KUKA KRL program: AM001.src, AM001.dat

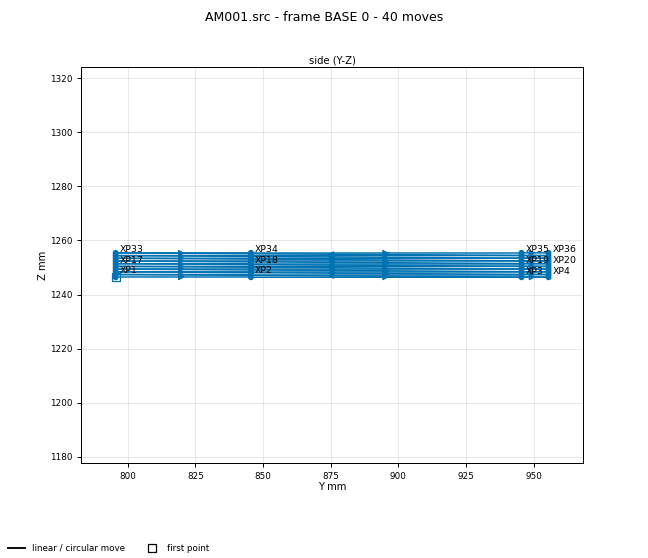
[picture p0: tool path of AM001.src in frame BASE 0, 40 of 42 moves have a stored position in this frame; points joined in program order, loops and branches not executed]
--- AM001.src ---
&ACCESS RVP
&REL 154
&PARAM TEMPLATE = C:\KRC\Roboter\Template\vorgabe
&PARAM EDITMASK = *
DEF AM001( )
;FOLD INI
  ;FOLD BASISTECH INI
    GLOBAL INTERRUPT DECL 3 WHEN $STOPMESS==TRUE DO IR_STOPM ( )
    INTERRUPT ON 3
    BAS (#INITMOV,0 )
  ;ENDFOLD (BASISTECH INI)
  ;FOLD USER INI
    ;Make your modifications here

  ;ENDFOLD (USER INI)
;ENDFOLD (INI)

;FOLD PTP HOME Vel=10 % DEFAULT;%{PE}%R 5.6.13,%MKUKATPBASIS,%CMOVE,%VPTP,%P 1:PTP, 2:HOME, 3:, 5:10, 7:DEFAULT
$BWDSTART=FALSE
PDAT_ACT=PDEFAULT
FDAT_ACT=FHOME
BAS(#PTP_PARAMS,10)
$H_POS=XHOME
PTP XHOME
;ENDFOLD

;FOLD OUT 33 'Gas 1' State=TRUE CONT;%{PE}%R 5.6.13,%MKUKATPBASIS,%COUT,%VOUTX,%P 2:33, 3:Gas 1, 5:TRUE, 6:CONTINUE
CONTINUE
$OUT[33]=TRUE
;ENDFOLD
;FOLD OUT 36 'Gas 2' State=TRUE CONT;%{PE}%R 5.6.13,%MKUKATPBASIS,%COUT,%VOUTX,%P 2:36, 3:Gas 2, 5:TRUE, 6:CONTINUE
CONTINUE
$OUT[36]=TRUE
;ENDFOLD
;FOLD WAIT Time=3 sec;%{PE}%R 5.6.13,%MKUKATPBASIS,%CWAIT,%VWAIT,%P 2:3
WAIT SEC 3
;ENDFOLD
;FOLD ANOUT POWDER=0.2 ;%{PE}%R 5.6.13,%MKUKATPBASIS,%CANA,%VANOUT_STAT,%P 2:CHANNEL_1, 4:0.2
$ANOUT[1]=0.2
;ENDFOLD
;FOLD LIN P1 Vel=0.035 m/s CPDAT1 Tool[1] Base[0];%{PE}%R 5.6.13,%MKUKATPBASIS,%CMOVE,%VLIN,%P 1:LIN, 2:P1, 3:, 5:0.035, 7:CPDAT1
$BWDSTART=FALSE
LDAT_ACT=LCPDAT1
FDAT_ACT=FP1
BAS(#CP_PARAMS,0.035)
LIN XP1
;ENDFOLD
;FOLD LIN P2 CONT Vel=0.035 m/s CPDAT2 Tool[1] Base[0];%{PE}%R 5.6.13,%MKUKATPBASIS,%CMOVE,%VLIN,%P 1:LIN, 2:P2, 3:C_DIS, 5:0.035, 7:CPDAT2
$BWDSTART=FALSE
LDAT_ACT=LCPDAT2
FDAT_ACT=FP2
BAS(#CP_PARAMS,0.035)
LIN XP2 C_DIS
;ENDFOLD
;FOLD SYN OUT 34 'Laser Shutter' State=TRUE at START Delay=0 ms;%{PE}%R 5.6.13,%MKUKATPBASIS,%COUT,%VSYNOUT,%P 2:34, 3:Laser Shutter, 5:TRUE, 7:0, 9:0, 12:0
TRIGGER WHEN DISTANCE=0 DELAY=0 DO $OUT[34]=TRUE
;ENDFOLD
;FOLD LIN P3 CONT Vel=0.035 m/s CPDAT3 Tool[1] Base[0];%{PE}%R 5.6.13,%MKUKATPBASIS,%CMOVE,%VLIN,%P 1:LIN, 2:P3, 3:C_DIS, 5:0.035, 7:CPDAT3
$BWDSTART=FALSE
LDAT_ACT=LCPDAT3
FDAT_ACT=FP3
BAS(#CP_PARAMS,0.035)
LIN XP3 C_DIS
;ENDFOLD
;FOLD SYN OUT 34 'Laser Shutter' State=FALSE at START Delay=0 ms;%{PE}%R 5.6.13,%MKUKATPBASIS,%COUT,%VSYNOUT,%P 2:34, 3:Laser Shutter, 5:FALSE, 7:0, 9:0, 12:0
TRIGGER WHEN DISTANCE=0 DELAY=0 DO $OUT[34]=FALSE
;ENDFOLD
;FOLD ANOUT POWDER=0 ;%{PE}%R 5.6.13,%MKUKATPBASIS,%CANA,%VANOUT_STAT,%P 2:CHANNEL_1, 4:0
$ANOUT[1]=0
;ENDFOLD
;FOLD LIN P4 Vel=0.035 m/s CPDAT4 Tool[1] Base[0];%{PE}%R 5.6.13,%MKUKATPBASIS,%CMOVE,%VLIN,%P 1:LIN, 2:P4, 3:, 5:0.035, 7:CPDAT4
$BWDSTART=FALSE
LDAT_ACT=LCPDAT4
FDAT_ACT=FP4
BAS(#CP_PARAMS,0.035)
LIN XP4
;ENDFOLD
;FOLD WAIT Time=0.1 sec;%{PE}%R 5.6.13,%MKUKATPBASIS,%CWAIT,%VWAIT,%P 2:0.1
WAIT SEC 0.1
;ENDFOLD
;FOLD ANOUT POWDER=0.2 ;%{PE}%R 5.6.13,%MKUKATPBASIS,%CANA,%VANOUT_STAT,%P 2:CHANNEL_1, 4:0.2
$ANOUT[1]=0.2
;ENDFOLD
;FOLD LIN P5 Vel=0.035 m/s CPDAT5 Tool[1] Base[0];%{PE}%R 5.6.13,%MKUKATPBASIS,%CMOVE,%VLIN,%P 1:LIN, 2:P5, 3:, 5:0.035, 7:CPDAT5
$BWDSTART=FALSE
LDAT_ACT=LCPDAT5
FDAT_ACT=FP5
BAS(#CP_PARAMS,0.035)
LIN XP5
;ENDFOLD
;FOLD LIN P6 CONT Vel=0.035 m/s CPDAT6 Tool[1] Base[0];%{PE}%R 5.6.13,%MKUKATPBASIS,%CMOVE,%VLIN,%P 1:LIN, 2:P6, 3:C_DIS, 5:0.035, 7:CPDAT6
$BWDSTART=FALSE
LDAT_ACT=LCPDAT6
FDAT_ACT=FP6
BAS(#CP_PARAMS,0.035)
LIN XP6 C_DIS
;ENDFOLD
;FOLD SYN OUT 34 'Laser Shutter' State=TRUE at START Delay=0 ms;%{PE}%R 5.6.13,%MKUKATPBASIS,%COUT,%VSYNOUT,%P 2:34, 3:Laser Shutter, 5:TRUE, 7:0, 9:0, 12:0
TRIGGER WHEN DISTANCE=0 DELAY=0 DO $OUT[34]=TRUE
;ENDFOLD
;FOLD LIN P7 CONT Vel=0.035 m/s CPDAT7 Tool[1] Base[0];%{PE}%R 5.6.13,%MKUKATPBASIS,%CMOVE,%VLIN,%P 1:LIN, 2:P7, 3:C_DIS, 5:0.035, 7:CPDAT7
$BWDSTART=FALSE
LDAT_ACT=LCPDAT7
FDAT_ACT=FP7
BAS(#CP_PARAMS,0.035)
LIN XP7 C_DIS
;ENDFOLD
;FOLD SYN OUT 34 'Laser Shutter' State=FALSE at START Delay=0 ms;%{PE}%R 5.6.13,%MKUKATPBASIS,%COUT,%VSYNOUT,%P 2:34, 3:Laser Shutter, 5:FALSE, 7:0, 9:0, 12:0
TRIGGER WHEN DISTANCE=0 DELAY=0 DO $OUT[34]=FALSE
;ENDFOLD
;FOLD ANOUT POWDER=0 ;%{PE}%R 5.6.13,%MKUKATPBASIS,%CANA,%VANOUT_STAT,%P 2:CHANNEL_1, 4:0
$ANOUT[1]=0
;ENDFOLD
;FOLD LIN P8 Vel=0.035 m/s CPDAT8 Tool[1] Base[0];%{PE}%R 5.6.13,%MKUKATPBASIS,%CMOVE,%VLIN,%P 1:LIN, 2:P8, 3:, 5:0.035, 7:CPDAT8
$BWDSTART=FALSE
LDAT_ACT=LCPDAT8
FDAT_ACT=FP8
BAS(#CP_PARAMS,0.035)
LIN XP8
;ENDFOLD
;FOLD WAIT Time=0.1 sec;%{PE}%R 5.6.13,%MKUKATPBASIS,%CWAIT,%VWAIT,%P 2:0.1
WAIT SEC 0.1
;ENDFOLD
;FOLD ANOUT POWDER=0.2 ;%{PE}%R 5.6.13,%MKUKATPBASIS,%CANA,%VANOUT_STAT,%P 2:CHANNEL_1, 4:0.2
$ANOUT[1]=0.2
;ENDFOLD
;FOLD LIN P9 Vel=0.035 m/s CPDAT9 Tool[1] Base[0];%{PE}%R 5.6.13,%MKUKATPBASIS,%CMOVE,%VLIN,%P 1:LIN, 2:P9, 3:, 5:0.035, 7:CPDAT9
$BWDSTART=FALSE
LDAT_ACT=LCPDAT9
FDAT_ACT=FP9
BAS(#CP_PARAMS,0.035)
LIN XP9
;ENDFOLD
;FOLD LIN P10 CONT Vel=0.035 m/s CPDAT10 Tool[1] Base[0];%{PE}%R 5.6.13,%MKUKATPBASIS,%CMOVE,%VLIN,%P 1:LIN, 2:P10, 3:C_DIS, 5:0.035, 7:CPDAT10
$BWDSTART=FALSE
LDAT_ACT=LCPDAT10
FDAT_ACT=FP10
BAS(#CP_PARAMS,0.035)
LIN XP10 C_DIS
;ENDFOLD
;FOLD SYN OUT 34 'Laser Shutter' State=TRUE at START Delay=0 ms;%{PE}%R 5.6.13,%MKUKATPBASIS,%COUT,%VSYNOUT,%P 2:34, 3:Laser Shutter, 5:TRUE, 7:0, 9:0, 12:0
TRIGGER WHEN DISTANCE=0 DELAY=0 DO $OUT[34]=TRUE
;ENDFOLD
;FOLD LIN P11 CONT Vel=0.035 m/s CPDAT11 Tool[1] Base[0];%{PE}%R 5.6.13,%MKUKATPBASIS,%CMOVE,%VLIN,%P 1:LIN, 2:P11, 3:C_DIS, 5:0.035, 7:CPDAT11
$BWDSTART=FALSE
LDAT_ACT=LCPDAT11
FDAT_ACT=FP11
BAS(#CP_PARAMS,0.035)
LIN XP11 C_DIS
;ENDFOLD
;FOLD SYN OUT 34 'Laser Shutter' State=FALSE at START Delay=0 ms;%{PE}%R 5.6.13,%MKUKATPBASIS,%COUT,%VSYNOUT,%P 2:34, 3:Laser Shutter, 5:FALSE, 7:0, 9:0, 12:0
TRIGGER WHEN DISTANCE=0 DELAY=0 DO $OUT[34]=FALSE
;ENDFOLD
;FOLD ANOUT POWDER=0 ;%{PE}%R 5.6.13,%MKUKATPBASIS,%CANA,%VANOUT_STAT,%P 2:CHANNEL_1, 4:0
$ANOUT[1]=0
;ENDFOLD
;FOLD LIN P12 Vel=0.035 m/s CPDAT12 Tool[1] Base[0];%{PE}%R 5.6.13,%MKUKATPBASIS,%CMOVE,%VLIN,%P 1:LIN, 2:P12, 3:, 5:0.035, 7:CPDAT12
$BWDSTART=FALSE
LDAT_ACT=LCPDAT12
FDAT_ACT=FP12
BAS(#CP_PARAMS,0.035)
LIN XP12
;ENDFOLD
;FOLD WAIT Time=0.1 sec;%{PE}%R 5.6.13,%MKUKATPBASIS,%CWAIT,%VWAIT,%P 2:0.1
WAIT SEC 0.1
;ENDFOLD
;FOLD ANOUT POWDER=0.2 ;%{PE}%R 5.6.13,%MKUKATPBASIS,%CANA,%VANOUT_STAT,%P 2:CHANNEL_1, 4:0.2
$ANOUT[1]=0.2
;ENDFOLD
;FOLD LIN P13 Vel=0.035 m/s CPDAT13 Tool[1] Base[0];%{PE}%R 5.6.13,%MKUKATPBASIS,%CMOVE,%VLIN,%P 1:LIN, 2:P13, 3:, 5:0.035, 7:CPDAT13
$BWDSTART=FALSE
LDAT_ACT=LCPDAT13
FDAT_ACT=FP13
BAS(#CP_PARAMS,0.035)
LIN XP13
;ENDFOLD
;FOLD LIN P14 CONT Vel=0.035 m/s CPDAT14 Tool[1] Base[0];%{PE}%R 5.6.13,%MKUKATPBASIS,%CMOVE,%VLIN,%P 1:LIN, 2:P14, 3:C_DIS, 5:0.035, 7:CPDAT14
$BWDSTART=FALSE
LDAT_ACT=LCPDAT14
FDAT_ACT=FP14
BAS(#CP_PARAMS,0.035)
LIN XP14 C_DIS
;ENDFOLD
;FOLD SYN OUT 34 'Laser Shutter' State=TRUE at START Delay=0 ms;%{PE}%R 5.6.13,%MKUKATPBASIS,%COUT,%VSYNOUT,%P 2:34, 3:Laser Shutter, 5:TRUE, 7:0, 9:0, 12:0
TRIGGER WHEN DISTANCE=0 DELAY=0 DO $OUT[34]=TRUE
;ENDFOLD
;FOLD LIN P15 CONT Vel=0.035 m/s CPDAT15 Tool[1] Base[0];%{PE}%R 5.6.13,%MKUKATPBASIS,%CMOVE,%VLIN,%P 1:LIN, 2:P15, 3:C_DIS, 5:0.035, 7:CPDAT15
$BWDSTART=FALSE
LDAT_ACT=LCPDAT15
FDAT_ACT=FP15
BAS(#CP_PARAMS,0.035)
LIN XP15 C_DIS
;ENDFOLD
;FOLD SYN OUT 34 'Laser Shutter' State=FALSE at START Delay=0 ms;%{PE}%R 5.6.13,%MKUKATPBASIS,%COUT,%VSYNOUT,%P 2:34, 3:Laser Shutter, 5:FALSE, 7:0, 9:0, 12:0
TRIGGER WHEN DISTANCE=0 DELAY=0 DO $OUT[34]=FALSE
;ENDFOLD
;FOLD ANOUT POWDER=0 ;%{PE}%R 5.6.13,%MKUKATPBASIS,%CANA,%VANOUT_STAT,%P 2:CHANNEL_1, 4:0
$ANOUT[1]=0
;ENDFOLD
;FOLD LIN P16 Vel=0.035 m/s CPDAT16 Tool[1] Base[0];%{PE}%R 5.6.13,%MKUKATPBASIS,%CMOVE,%VLIN,%P 1:LIN, 2:P16, 3:, 5:0.035, 7:CPDAT16
$BWDSTART=FALSE
LDAT_ACT=LCPDAT16
FDAT_ACT=FP16
BAS(#CP_PARAMS,0.035)
LIN XP16
;ENDFOLD
;FOLD WAIT Time=0.1 sec;%{PE}%R 5.6.13,%MKUKATPBASIS,%CWAIT,%VWAIT,%P 2:0.1
WAIT SEC 0.1
;ENDFOLD
;FOLD ANOUT POWDER=0.2 ;%{PE}%R 5.6.13,%MKUKATPBASIS,%CANA,%VANOUT_STAT,%P 2:CHANNEL_1, 4:0.2
$ANOUT[1]=0.2
;ENDFOLD
;FOLD LIN P17 Vel=0.035 m/s CPDAT17 Tool[1] Base[0];%{PE}%R 5.6.13,%MKUKATPBASIS,%CMOVE,%VLIN,%P 1:LIN, 2:P17, 3:, 5:0.035, 7:CPDAT17
$BWDSTART=FALSE
LDAT_ACT=LCPDAT17
FDAT_ACT=FP17
BAS(#CP_PARAMS,0.035)
LIN XP17
;ENDFOLD
;FOLD LIN P18 CONT Vel=0.035 m/s CPDAT18 Tool[1] Base[0];%{PE}%R 5.6.13,%MKUKATPBASIS,%CMOVE,%VLIN,%P 1:LIN, 2:P18, 3:C_DIS, 5:0.035, 7:CPDAT18
$BWDSTART=FALSE
LDAT_ACT=LCPDAT18
FDAT_ACT=FP18
BAS(#CP_PARAMS,0.035)
LIN XP18 C_DIS
;ENDFOLD
;FOLD SYN OUT 34 'Laser Shutter' State=TRUE at START Delay=0 ms;%{PE}%R 5.6.13,%MKUKATPBASIS,%COUT,%VSYNOUT,%P 2:34, 3:Laser Shutter, 5:TRUE, 7:0, 9:0, 12:0
TRIGGER WHEN DISTANCE=0 DELAY=0 DO $OUT[34]=TRUE
;ENDFOLD
;FOLD LIN P19 CONT Vel=0.035 m/s CPDAT19 Tool[1] Base[0];%{PE}%R 5.6.13,%MKUKATPBASIS,%CMOVE,%VLIN,%P 1:LIN, 2:P19, 3:C_DIS, 5:0.035, 7:CPDAT19
$BWDSTART=FALSE
LDAT_ACT=LCPDAT19
FDAT_ACT=FP19
BAS(#CP_PARAMS,0.035)
LIN XP19 C_DIS
;ENDFOLD
;FOLD SYN OUT 34 'Laser Shutter' State=FALSE at START Delay=0 ms;%{PE}%R 5.6.13,%MKUKATPBASIS,%COUT,%VSYNOUT,%P 2:34, 3:Laser Shutter, 5:FALSE, 7:0, 9:0, 12:0
TRIGGER WHEN DISTANCE=0 DELAY=0 DO $OUT[34]=FALSE
;ENDFOLD
;FOLD ANOUT POWDER=0 ;%{PE}%R 5.6.13,%MKUKATPBASIS,%CANA,%VANOUT_STAT,%P 2:CHANNEL_1, 4:0
$ANOUT[1]=0
;ENDFOLD
;FOLD LIN P20 Vel=0.035 m/s CPDAT20 Tool[1] Base[0];%{PE}%R 5.6.13,%MKUKATPBASIS,%CMOVE,%VLIN,%P 1:LIN, 2:P20, 3:, 5:0.035, 7:CPDAT20
$BWDSTART=FALSE
LDAT_ACT=LCPDAT20
FDAT_ACT=FP20
BAS(#CP_PARAMS,0.035)
LIN XP20
;ENDFOLD
;FOLD WAIT Time=0.1 sec;%{PE}%R 5.6.13,%MKUKATPBASIS,%CWAIT,%VWAIT,%P 2:0.1
WAIT SEC 0.1
;ENDFOLD
;FOLD ANOUT POWDER=0.2 ;%{PE}%R 5.6.13,%MKUKATPBASIS,%CANA,%VANOUT_STAT,%P 2:CHANNEL_1, 4:0.2
$ANOUT[1]=0.2
;ENDFOLD
;FOLD LIN P21 Vel=0.035 m/s CPDAT21 Tool[1] Base[0];%{PE}%R 5.6.13,%MKUKATPBASIS,%CMOVE,%VLIN,%P 1:LIN, 2:P21, 3:, 5:0.035, 7:CPDAT21
$BWDSTART=FALSE
LDAT_ACT=LCPDAT21
FDAT_ACT=FP21
BAS(#CP_PARAMS,0.035)
LIN XP21
;ENDFOLD
;FOLD LIN P22 CONT Vel=0.035 m/s CPDAT22 Tool[1] Base[0];%{PE}%R 5.6.13,%MKUKATPBASIS,%CMOVE,%VLIN,%P 1:LIN, 2:P22, 3:C_DIS, 5:0.035, 7:CPDAT22
$BWDSTART=FALSE
LDAT_ACT=LCPDAT22
FDAT_ACT=FP22
BAS(#CP_PARAMS,0.035)
LIN XP22 C_DIS
;ENDFOLD
;FOLD SYN OUT 34 'Laser Shutter' State=TRUE at START Delay=0 ms;%{PE}%R 5.6.13,%MKUKATPBASIS,%COUT,%VSYNOUT,%P 2:34, 3:Laser Shutter, 5:TRUE, 7:0, 9:0, 12:0
TRIGGER WHEN DISTANCE=0 DELAY=0 DO $OUT[34]=TRUE
;ENDFOLD
;FOLD LIN P23 CONT Vel=0.035 m/s CPDAT23 Tool[1] Base[0];%{PE}%R 5.6.13,%MKUKATPBASIS,%CMOVE,%VLIN,%P 1:LIN, 2:P23, 3:C_DIS, 5:0.035, 7:CPDAT23
$BWDSTART=FALSE
LDAT_ACT=LCPDAT23
FDAT_ACT=FP23
BAS(#CP_PARAMS,0.035)
LIN XP23 C_DIS
;ENDFOLD
;FOLD SYN OUT 34 'Laser Shutter' State=FALSE at START Delay=0 ms;%{PE}%R 5.6.13,%MKUKATPBASIS,%COUT,%VSYNOUT,%P 2:34, 3:Laser Shutter, 5:FALSE, 7:0, 9:0, 12:0
TRIGGER WHEN DISTANCE=0 DELAY=0 DO $OUT[34]=FALSE
;ENDFOLD
;FOLD ANOUT POWDER=0 ;%{PE}%R 5.6.13,%MKUKATPBASIS,%CANA,%VANOUT_STAT,%P 2:CHANNEL_1, 4:0
$ANOUT[1]=0
;ENDFOLD
;FOLD LIN P24 Vel=0.035 m/s CPDAT24 Tool[1] Base[0];%{PE}%R 5.6.13,%MKUKATPBASIS,%CMOVE,%VLIN,%P 1:LIN, 2:P24, 3:, 5:0.035, 7:CPDAT24
$BWDSTART=FALSE
LDAT_ACT=LCPDAT24
FDAT_ACT=FP24
BAS(#CP_PARAMS,0.035)
LIN XP24
;ENDFOLD
;FOLD WAIT Time=0.1 sec;%{PE}%R 5.6.13,%MKUKATPBASIS,%CWAIT,%VWAIT,%P 2:0.1
WAIT SEC 0.1
;ENDFOLD
;FOLD ANOUT POWDER=0.2 ;%{PE}%R 5.6.13,%MKUKATPBASIS,%CANA,%VANOUT_STAT,%P 2:CHANNEL_1, 4:0.2
$ANOUT[1]=0.2
;ENDFOLD
;FOLD LIN P25 Vel=0.035 m/s CPDAT25 Tool[1] Base[0];%{PE}%R 5.6.13,%MKUKATPBASIS,%CMOVE,%VLIN,%P 1:LIN, 2:P25, 3:, 5:0.035, 7:CPDAT25
$BWDSTART=FALSE
LDAT_ACT=LCPDAT25
FDAT_ACT=FP25
BAS(#CP_PARAMS,0.035)
LIN XP25
;ENDFOLD
;FOLD LIN P26 CONT Vel=0.035 m/s CPDAT26 Tool[1] Base[0];%{PE}%R 5.6.13,%MKUKATPBASIS,%CMOVE,%VLIN,%P 1:LIN, 2:P26, 3:C_DIS, 5:0.035, 7:CPDAT26
$BWDSTART=FALSE
LDAT_ACT=LCPDAT26
FDAT_ACT=FP26
BAS(#CP_PARAMS,0.035)
LIN XP26 C_DIS
;ENDFOLD
;FOLD SYN OUT 34 'Laser Shutter' State=TRUE at START Delay=0 ms;%{PE}%R 5.6.13,%MKUKATPBASIS,%COUT,%VSYNOUT,%P 2:34, 3:Laser Shutter, 5:TRUE, 7:0, 9:0, 12:0
TRIGGER WHEN DISTANCE=0 DELAY=0 DO $OUT[34]=TRUE
;ENDFOLD
;FOLD LIN P27 CONT Vel=0.035 m/s CPDAT27 Tool[1] Base[0];%{PE}%R 5.6.13,%MKUKATPBASIS,%CMOVE,%VLIN,%P 1:LIN, 2:P27, 3:C_DIS, 5:0.035, 7:CPDAT27
$BWDSTART=FALSE
LDAT_ACT=LCPDAT27
FDAT_ACT=FP27
BAS(#CP_PARAMS,0.035)
LIN XP27 C_DIS
;ENDFOLD
;FOLD SYN OUT 34 'Laser Shutter' State=FALSE at START Delay=0 ms;%{PE}%R 5.6.13,%MKUKATPBASIS,%COUT,%VSYNOUT,%P 2:34, 3:Laser Shutter, 5:FALSE, 7:0, 9:0, 12:0
TRIGGER WHEN DISTANCE=0 DELAY=0 DO $OUT[34]=FALSE
;ENDFOLD
;FOLD ANOUT POWDER=0 ;%{PE}%R 5.6.13,%MKUKATPBASIS,%CANA,%VANOUT_STAT,%P 2:CHANNEL_1, 4:0
$ANOUT[1]=0
;ENDFOLD
;FOLD LIN P28 Vel=0.035 m/s CPDAT28 Tool[1] Base[0];%{PE}%R 5.6.13,%MKUKATPBASIS,%CMOVE,%VLIN,%P 1:LIN, 2:P28, 3:, 5:0.035, 7:CPDAT28
$BWDSTART=FALSE
LDAT_ACT=LCPDAT28
FDAT_ACT=FP28
BAS(#CP_PARAMS,0.035)
LIN XP28
;ENDFOLD
;FOLD WAIT Time=0.1 sec;%{PE}%R 5.6.13,%MKUKATPBASIS,%CWAIT,%VWAIT,%P 2:0.1
WAIT SEC 0.1
;ENDFOLD
;FOLD ANOUT POWDER=0.2 ;%{PE}%R 5.6.13,%MKUKATPBASIS,%CANA,%VANOUT_STAT,%P 2:CHANNEL_1, 4:0.2
$ANOUT[1]=0.2
;ENDFOLD
;FOLD LIN P29 Vel=0.035 m/s CPDAT29 Tool[1] Base[0];%{PE}%R 5.6.13,%MKUKATPBASIS,%CMOVE,%VLIN,%P 1:LIN, 2:P29, 3:, 5:0.035, 7:CPDAT29
$BWDSTART=FALSE
LDAT_ACT=LCPDAT29
FDAT_ACT=FP29
BAS(#CP_PARAMS,0.035)
LIN XP29
;ENDFOLD
;FOLD LIN P30 CONT Vel=0.035 m/s CPDAT30 Tool[1] Base[0];%{PE}%R 5.6.13,%MKUKATPBASIS,%CMOVE,%VLIN,%P 1:LIN, 2:P30, 3:C_DIS, 5:0.035, 7:CPDAT30
$BWDSTART=FALSE
LDAT_ACT=LCPDAT30
FDAT_ACT=FP30
BAS(#CP_PARAMS,0.035)
LIN XP30 C_DIS
;ENDFOLD
;FOLD SYN OUT 34 'Laser Shutter' State=TRUE at START Delay=0 ms;%{PE}%R 5.6.13,%MKUKATPBASIS,%COUT,%VSYNOUT,%P 2:34, 3:Laser Shutter, 5:TRUE, 7:0, 9:0, 12:0
TRIGGER WHEN DISTANCE=0 DELAY=0 DO $OUT[34]=TRUE
;ENDFOLD
;FOLD LIN P31 CONT Vel=0.035 m/s CPDAT31 Tool[1] Base[0];%{PE}%R 5.6.13,%MKUKATPBASIS,%CMOVE,%VLIN,%P 1:LIN, 2:P31, 3:C_DIS, 5:0.035, 7:CPDAT31
$BWDSTART=FALSE
LDAT_ACT=LCPDAT31
FDAT_ACT=FP31
BAS(#CP_PARAMS,0.035)
LIN XP31 C_DIS
;ENDFOLD
;FOLD SYN OUT 34 'Laser Shutter' State=FALSE at START Delay=0 ms;%{PE}%R 5.6.13,%MKUKATPBASIS,%COUT,%VSYNOUT,%P 2:34, 3:Laser Shutter, 5:FALSE, 7:0, 9:0, 12:0
TRIGGER WHEN DISTANCE=0 DELAY=0 DO $OUT[34]=FALSE
;ENDFOLD
;FOLD ANOUT POWDER=0 ;%{PE}%R 5.6.13,%MKUKATPBASIS,%CANA,%VANOUT_STAT,%P 2:CHANNEL_1, 4:0
$ANOUT[1]=0
;ENDFOLD
;FOLD LIN P32 Vel=0.035 m/s CPDAT32 Tool[1] Base[0];%{PE}%R 5.6.13,%MKUKATPBASIS,%CMOVE,%VLIN,%P 1:LIN, 2:P32, 3:, 5:0.035, 7:CPDAT32
$BWDSTART=FALSE
LDAT_ACT=LCPDAT32
FDAT_ACT=FP32
BAS(#CP_PARAMS,0.035)
LIN XP32
;ENDFOLD
;FOLD WAIT Time=0.1 sec;%{PE}%R 5.6.13,%MKUKATPBASIS,%CWAIT,%VWAIT,%P 2:0.1
WAIT SEC 0.1
;ENDFOLD
;FOLD ANOUT POWDER=0.2 ;%{PE}%R 5.6.13,%MKUKATPBASIS,%CANA,%VANOUT_STAT,%P 2:CHANNEL_1, 4:0.2
$ANOUT[1]=0.2
;ENDFOLD
;FOLD LIN P33 Vel=0.035 m/s CPDAT33 Tool[1] Base[0];%{PE}%R 5.6.13,%MKUKATPBASIS,%CMOVE,%VLIN,%P 1:LIN, 2:P33, 3:, 5:0.035, 7:CPDAT33
$BWDSTART=FALSE
LDAT_ACT=LCPDAT33
FDAT_ACT=FP33
BAS(#CP_PARAMS,0.035)
LIN XP33
;ENDFOLD
;FOLD LIN P34 CONT Vel=0.035 m/s CPDAT34 Tool[1] Base[0];%{PE}%R 5.6.13,%MKUKATPBASIS,%CMOVE,%VLIN,%P 1:LIN, 2:P34, 3:C_DIS, 5:0.035, 7:CPDAT34
$BWDSTART=FALSE
LDAT_ACT=LCPDAT34
FDAT_ACT=FP34
BAS(#CP_PARAMS,0.035)
LIN XP34 C_DIS
;ENDFOLD
;FOLD SYN OUT 34 'Laser Shutter' State=TRUE at START Delay=0 ms;%{PE}%R 5.6.13,%MKUKATPBASIS,%COUT,%VSYNOUT,%P 2:34, 3:Laser Shutter, 5:TRUE, 7:0, 9:0, 12:0
TRIGGER WHEN DISTANCE=0 DELAY=0 DO $OUT[34]=TRUE
;ENDFOLD
;FOLD LIN P35 CONT Vel=0.035 m/s CPDAT35 Tool[1] Base[0];%{PE}%R 5.6.13,%MKUKATPBASIS,%CMOVE,%VLIN,%P 1:LIN, 2:P35, 3:C_DIS, 5:0.035, 7:CPDAT35
$BWDSTART=FALSE
LDAT_ACT=LCPDAT35
FDAT_ACT=FP35
BAS(#CP_PARAMS,0.035)
LIN XP35 C_DIS
;ENDFOLD
;FOLD SYN OUT 34 'Laser Shutter' State=FALSE at START Delay=0 ms;%{PE}%R 5.6.13,%MKUKATPBASIS,%COUT,%VSYNOUT,%P 2:34, 3:Laser Shutter, 5:FALSE, 7:0, 9:0, 12:0
TRIGGER WHEN DISTANCE=0 DELAY=0 DO $OUT[34]=FALSE
;ENDFOLD
;FOLD ANOUT POWDER=0 ;%{PE}%R 5.6.13,%MKUKATPBASIS,%CANA,%VANOUT_STAT,%P 2:CHANNEL_1, 4:0
$ANOUT[1]=0
;ENDFOLD
;FOLD LIN P36 Vel=0.035 m/s CPDAT36 Tool[1] Base[0];%{PE}%R 5.6.13,%MKUKATPBASIS,%CMOVE,%VLIN,%P 1:LIN, 2:P36, 3:, 5:0.035, 7:CPDAT36
$BWDSTART=FALSE
LDAT_ACT=LCPDAT36
FDAT_ACT=FP36
BAS(#CP_PARAMS,0.035)
LIN XP36
;ENDFOLD
;FOLD WAIT Time=0.1 sec;%{PE}%R 5.6.13,%MKUKATPBASIS,%CWAIT,%VWAIT,%P 2:0.1
WAIT SEC 0.1
;ENDFOLD
;FOLD ANOUT POWDER=0.2 ;%{PE}%R 5.6.13,%MKUKATPBASIS,%CANA,%VANOUT_STAT,%P 2:CHANNEL_1, 4:0.2
$ANOUT[1]=0.2
;ENDFOLD
;FOLD LIN P37 Vel=0.035 m/s CPDAT37 Tool[1] Base[0];%{PE}%R 5.6.13,%MKUKATPBASIS,%CMOVE,%VLIN,%P 1:LIN, 2:P37, 3:, 5:0.035, 7:CPDAT37
$BWDSTART=FALSE
LDAT_ACT=LCPDAT37
FDAT_ACT=FP37
BAS(#CP_PARAMS,0.035)
LIN XP37
;ENDFOLD
;FOLD LIN P38 CONT Vel=0.035 m/s CPDAT38 Tool[1] Base[0];%{PE}%R 5.6.13,%MKUKATPBASIS,%CMOVE,%VLIN,%P 1:LIN, 2:P38, 3:C_DIS, 5:0.035, 7:CPDAT38
$BWDSTART=FALSE
LDAT_ACT=LCPDAT38
FDAT_ACT=FP38
BAS(#CP_PARAMS,0.035)
LIN XP38 C_DIS
;ENDFOLD
;FOLD SYN OUT 34 'Laser Shutter' State=TRUE at START Delay=0 ms;%{PE}%R 5.6.13,%MKUKATPBASIS,%COUT,%VSYNOUT,%P 2:34, 3:Laser Shutter, 5:TRUE, 7:0, 9:0, 12:0
TRIGGER WHEN DISTANCE=0 DELAY=0 DO $OUT[34]=TRUE
;ENDFOLD
;FOLD LIN P39 CONT Vel=0.035 m/s CPDAT39 Tool[1] Base[0];%{PE}%R 5.6.13,%MKUKATPBASIS,%CMOVE,%VLIN,%P 1:LIN, 2:P39, 3:C_DIS, 5:0.035, 7:CPDAT39
$BWDSTART=FALSE
LDAT_ACT=LCPDAT39
FDAT_ACT=FP39
BAS(#CP_PARAMS,0.035)
LIN XP39 C_DIS
;ENDFOLD
;FOLD SYN OUT 34 'Laser Shutter' State=FALSE at START Delay=0 ms;%{PE}%R 5.6.13,%MKUKATPBASIS,%COUT,%VSYNOUT,%P 2:34, 3:Laser Shutter, 5:FALSE, 7:0, 9:0, 12:0
TRIGGER WHEN DISTANCE=0 DELAY=0 DO $OUT[34]=FALSE
;ENDFOLD
;FOLD ANOUT POWDER=0 ;%{PE}%R 5.6.13,%MKUKATPBASIS,%CANA,%VANOUT_STAT,%P 2:CHANNEL_1, 4:0
$ANOUT[1]=0
;ENDFOLD
;FOLD LIN P40 Vel=0.035 m/s CPDAT40 Tool[1] Base[0];%{PE}%R 5.6.13,%MKUKATPBASIS,%CMOVE,%VLIN,%P 1:LIN, 2:P40, 3:, 5:0.035, 7:CPDAT40
$BWDSTART=FALSE
LDAT_ACT=LCPDAT40
FDAT_ACT=FP40
BAS(#CP_PARAMS,0.035)
LIN XP40
;ENDFOLD
;FOLD OUT 33 'Gas 1' State=FALSE CONT;%{PE}%R 5.6.13,%MKUKATPBASIS,%COUT,%VOUTX,%P 2:33, 3:Gas 1, 5:FALSE, 6:CONTINUE
CONTINUE
$OUT[33]=FALSE
;ENDFOLD
;FOLD OUT 36 'Gas 2' State=FALSE CONT;%{PE}%R 5.6.13,%MKUKATPBASIS,%COUT,%VOUTX,%P 2:36, 3:Gas 2, 5:FALSE, 6:CONTINUE
CONTINUE
$OUT[36]=FALSE
;ENDFOLD
;FOLD WAIT Time=0.1 sec;%{PE}%R 5.6.13,%MKUKATPBASIS,%CWAIT,%VWAIT,%P 2:0.1
WAIT SEC 0.1
;ENDFOLD
;FOLD PTP HOME Vel=10 % DEFAULT;%{PE}%R 5.6.13,%MKUKATPBASIS,%CMOVE,%VPTP,%P 1:PTP, 2:HOME, 3:, 5:10, 7:DEFAULT
$BWDSTART=FALSE
PDAT_ACT=PDEFAULT
FDAT_ACT=FHOME
BAS(#PTP_PARAMS,10)
$H_POS=XHOME
PTP XHOME
;ENDFOLD

END

--- AM001.dat ---
&ACCESS RVP
&REL 154
&PARAM TEMPLATE = C:\KRC\Roboter\Template\vorgabe
&PARAM EDITMASK = *
DEFDAT  AM001
;FOLD EXTERNAL DECLARATIONS;%{PE}%MKUKATPBASIS,%CEXT,%VCOMMON,%P
;FOLD BASISTECH EXT;%{PE}%MKUKATPBASIS,%CEXT,%VEXT,%P
EXT  BAS (BAS_COMMAND  :IN,REAL  :IN )
DECL INT SUCCESS
;ENDFOLD (BASISTECH EXT)
;FOLD USER EXT;%{E}%MKUKATPUSER,%CEXT,%VEXT,%P
;Make here your modifications

;ENDFOLD (USER EXT)
;ENDFOLD (EXTERNAL DECLARATIONS)
DECL BASIS_SUGG_T LAST_BASIS={POINT1[] "P40                     ",POINT2[] "P40                     ",CP_PARAMS[] "CPDAT40                 ",PTP_PARAMS[] "PDAT0                   ",CONT[] "                        ",CP_VEL[] "0.035                   ",PTP_VEL[] "100                     ",SYNC_PARAMS[] "SYNCDAT                 ",SPL_NAME[] "S0                      "}
DECL E6POS XP1={X 984.658997,Y 795.544373,Z 1246.38501,A -157.893402,B 46.0296097,C -166.345901,S 2,T 35,E1 0.0,E2 0.0,E3 0.0,E4 0.0,E5 0.0,E6 0.0}
DECL FDAT FP1={TOOL_NO 1,BASE_NO 0,IPO_FRAME #BASE,POINT2[] " ",TQ_STATE FALSE}
DECL LDAT LCPDAT1={VEL 2.0,ACC 100.0,APO_DIST 100.0,APO_FAC 50.0,ORI_TYP #VAR,CIRC_TYP #BASE,JERK_FAC 50.0,EXAX_IGN 0}
DECL E6POS XP2={X 984.658691,Y 845.544922,Z 1246.38501,A -157.894394,B 46.0297585,C -166.346298,S 2,T 35,E1 0.0,E2 0.0,E3 0.0,E4 0.0,E5 0.0,E6 0.0}
DECL FDAT FP2={TOOL_NO 1,BASE_NO 0,IPO_FRAME #BASE,POINT2[] " ",TQ_STATE FALSE}
DECL LDAT LCPDAT2={VEL 2.0,ACC 100.0,APO_DIST 100.0,APO_FAC 50.0,ORI_TYP #VAR,CIRC_TYP #BASE,JERK_FAC 50.0,EXAX_IGN 0}
DECL E6POS XP3={X 984.660217,Y 945.544373,Z 1246.38098,A -157.894699,B 46.0296402,C -166.346298,S 2,T 35,E1 0.0,E2 0.0,E3 0.0,E4 0.0,E5 0.0,E6 0.0}
DECL FDAT FP3={TOOL_NO 1,BASE_NO 0,IPO_FRAME #BASE,POINT2[] " ",TQ_STATE FALSE}
DECL LDAT LCPDAT3={VEL 2.0,ACC 100.0,APO_DIST 100.0,APO_FAC 50.0,ORI_TYP #VAR,CIRC_TYP #BASE,JERK_FAC 50.0,EXAX_IGN 0}
DECL E6POS XP4={X 984.660217,Y 955.543884,Z 1246.38098,A -157.895798,B 46.0295906,C -166.347,S 2,T 35,E1 0.0,E2 0.0,E3 0.0,E4 0.0,E5 0.0,E6 0.0}
DECL FDAT FP4={TOOL_NO 1,BASE_NO 0,IPO_FRAME #BASE,POINT2[] " ",TQ_STATE FALSE}
DECL LDAT LCPDAT4={VEL 2.0,ACC 100.0,APO_DIST 100.0,APO_FAC 50.0,ORI_TYP #VAR,CIRC_TYP #BASE,JERK_FAC 50.0,EXAX_IGN 0}
DECL E6POS XP5={X 984.658081,Y 795.542725,Z 1247.38794,A -157.895905,B 46.0301704,C -166.347397,S 2,T 35,E1 0.0,E2 0.0,E3 0.0,E4 0.0,E5 0.0,E6 0.0}
DECL FDAT FP5={TOOL_NO 1,BASE_NO 0,IPO_FRAME #BASE,POINT2[] " ",TQ_STATE FALSE}
DECL LDAT LCPDAT5={VEL 2.0,ACC 100.0,APO_DIST 100.0,APO_FAC 50.0,ORI_TYP #VAR,CIRC_TYP #BASE,JERK_FAC 50.0,EXAX_IGN 0}
DECL E6POS XP6={X 984.656006,Y 845.54657,Z 1247.38696,A -157.895401,B 46.029911,C -166.347305,S 2,T 35,E1 0.0,E2 0.0,E3 0.0,E4 0.0,E5 0.0,E6 0.0}
DECL FDAT FP6={TOOL_NO 1,BASE_NO 0,IPO_FRAME #BASE,POINT2[] " ",TQ_STATE FALSE}
DECL LDAT LCPDAT6={VEL 2.0,ACC 100.0,APO_DIST 100.0,APO_FAC 50.0,ORI_TYP #VAR,CIRC_TYP #BASE,JERK_FAC 50.0,EXAX_IGN 0}
DECL E6POS XP7={X 984.654419,Y 945.547974,Z 1247.38696,A -157.895996,B 46.0300407,C -166.347794,S 2,T 35,E1 0.0,E2 0.0,E3 0.0,E4 0.0,E5 0.0,E6 0.0}
DECL FDAT FP7={TOOL_NO 1,BASE_NO 0,IPO_FRAME #BASE,POINT2[] " ",TQ_STATE FALSE}
DECL LDAT LCPDAT7={VEL 2.0,ACC 100.0,APO_DIST 100.0,APO_FAC 50.0,ORI_TYP #VAR,CIRC_TYP #BASE,JERK_FAC 50.0,EXAX_IGN 0}
DECL E6POS XP8={X 984.659729,Y 955.543274,Z 1247.38403,A -157.896698,B 46.0294914,C -166.347504,S 2,T 35,E1 0.0,E2 0.0,E3 0.0,E4 0.0,E5 0.0,E6 0.0}
DECL FDAT FP8={TOOL_NO 1,BASE_NO 0,IPO_FRAME #BASE,POINT2[] " ",TQ_STATE FALSE}
DECL LDAT LCPDAT8={VEL 2.0,ACC 100.0,APO_DIST 100.0,APO_FAC 50.0,ORI_TYP #VAR,CIRC_TYP #BASE,JERK_FAC 50.0,EXAX_IGN 0}
DECL E6POS XP9={X 984.657776,Y 795.544128,Z 1248.38904,A -157.897003,B 46.0303497,C -166.348801,S 2,T 35,E1 0.0,E2 0.0,E3 0.0,E4 0.0,E5 0.0,E6 0.0}
DECL FDAT FP9={TOOL_NO 1,BASE_NO 0,IPO_FRAME #BASE,POINT2[] " ",TQ_STATE FALSE}
DECL LDAT LCPDAT9={VEL 2.0,ACC 100.0,APO_DIST 100.0,APO_FAC 50.0,ORI_TYP #VAR,CIRC_TYP #BASE,JERK_FAC 50.0,EXAX_IGN 0}
DECL E6POS XP10={X 984.655579,Y 845.546204,Z 1248.38696,A -157.894897,B 46.0300598,C -166.346893,S 2,T 35,E1 0.0,E2 0.0,E3 0.0,E4 0.0,E5 0.0,E6 0.0}
DECL FDAT FP10={TOOL_NO 1,BASE_NO 0,IPO_FRAME #BASE,POINT2[] " ",TQ_STATE FALSE}
DECL LDAT LCPDAT10={VEL 2.0,ACC 100.0,APO_DIST 100.0,APO_FAC 50.0,ORI_TYP #VAR,CIRC_TYP #BASE,JERK_FAC 50.0,EXAX_IGN 0}
DECL E6POS XP11={X 984.653625,Y 945.547485,Z 1248.38696,A -157.895996,B 46.0299988,C -166.3479,S 2,T 35,E1 0.0,E2 0.0,E3 0.0,E4 0.0,E5 0.0,E6 0.0}
DECL FDAT FP11={TOOL_NO 1,BASE_NO 0,IPO_FRAME #BASE,POINT2[] " ",TQ_STATE FALSE}
DECL LDAT LCPDAT11={VEL 2.0,ACC 100.0,APO_DIST 100.0,APO_FAC 50.0,ORI_TYP #VAR,CIRC_TYP #BASE,JERK_FAC 50.0,EXAX_IGN 0}
DECL E6POS XP12={X 984.663208,Y 955.538086,Z 1248.38501,A -157.8965,B 46.0294304,C -166.347,S 2,T 35,E1 0.0,E2 0.0,E3 0.0,E4 0.0,E5 0.0,E6 0.0}
DECL FDAT FP12={TOOL_NO 1,BASE_NO 0,IPO_FRAME #BASE,POINT2[] " ",TQ_STATE FALSE}
DECL LDAT LCPDAT12={VEL 2.0,ACC 100.0,APO_DIST 100.0,APO_FAC 50.0,ORI_TYP #VAR,CIRC_TYP #BASE,JERK_FAC 50.0,EXAX_IGN 0}
DECL E6POS XP13={X 984.656494,Y 795.544006,Z 1249.39001,A -157.897903,B 46.0304489,C -166.349701,S 2,T 35,E1 0.0,E2 0.0,E3 0.0,E4 0.0,E5 0.0,E6 0.0}
DECL FDAT FP13={TOOL_NO 1,BASE_NO 0,IPO_FRAME #BASE,POINT2[] " ",TQ_STATE FALSE}
DECL LDAT LCPDAT13={VEL 2.0,ACC 100.0,APO_DIST 100.0,APO_FAC 50.0,ORI_TYP #VAR,CIRC_TYP #BASE,JERK_FAC 50.0,EXAX_IGN 0}
DECL E6POS XP14={X 984.654785,Y 845.545105,Z 1249.39001,A -157.894897,B 46.0302391,C -166.346893,S 2,T 35,E1 0.0,E2 0.0,E3 0.0,E4 0.0,E5 0.0,E6 0.0}
DECL FDAT FP14={TOOL_NO 1,BASE_NO 0,IPO_FRAME #BASE,POINT2[] " ",TQ_STATE FALSE}
DECL LDAT LCPDAT14={VEL 2.0,ACC 100.0,APO_DIST 100.0,APO_FAC 50.0,ORI_TYP #VAR,CIRC_TYP #BASE,JERK_FAC 50.0,EXAX_IGN 0}
DECL E6POS XP15={X 984.655884,Y 945.544617,Z 1249.39099,A -157.895096,B 46.0303497,C -166.347,S 2,T 35,E1 0.0,E2 0.0,E3 0.0,E4 0.0,E5 0.0,E6 0.0}
DECL FDAT FP15={TOOL_NO 1,BASE_NO 0,IPO_FRAME #BASE,POINT2[] " ",TQ_STATE FALSE}
DECL LDAT LCPDAT15={VEL 2.0,ACC 100.0,APO_DIST 100.0,APO_FAC 50.0,ORI_TYP #VAR,CIRC_TYP #BASE,JERK_FAC 50.0,EXAX_IGN 0}
DECL E6POS XP16={X 984.661987,Y 955.536072,Z 1249.38696,A -157.897003,B 46.0292892,C -166.347107,S 2,T 35,E1 0.0,E2 0.0,E3 0.0,E4 0.0,E5 0.0,E6 0.0}
DECL FDAT FP16={TOOL_NO 1,BASE_NO 0,IPO_FRAME #BASE,POINT2[] " ",TQ_STATE FALSE}
DECL LDAT LCPDAT16={VEL 2.0,ACC 100.0,APO_DIST 100.0,APO_FAC 50.0,ORI_TYP #VAR,CIRC_TYP #BASE,JERK_FAC 50.0,EXAX_IGN 0}
DECL E6POS XP17={X 984.655518,Y 795.544678,Z 1250.38794,A -157.899094,B 46.0303192,C -166.350906,S 2,T 35,E1 0.0,E2 0.0,E3 0.0,E4 0.0,E5 0.0,E6 0.0}
DECL FDAT FP17={TOOL_NO 1,BASE_NO 0,IPO_FRAME #BASE,POINT2[] " ",TQ_STATE FALSE}
DECL LDAT LCPDAT17={VEL 2.0,ACC 100.0,APO_DIST 100.0,APO_FAC 50.0,ORI_TYP #VAR,CIRC_TYP #BASE,JERK_FAC 50.0,EXAX_IGN 0}
DECL E6POS XP18={X 984.651672,Y 845.546082,Z 1250.39502,A -157.893799,B 46.0302696,C -166.346298,S 2,T 35,E1 0.0,E2 0.0,E3 0.0,E4 0.0,E5 0.0,E6 0.0}
DECL FDAT FP18={TOOL_NO 1,BASE_NO 0,IPO_FRAME #BASE,POINT2[] " ",TQ_STATE FALSE}
DECL LDAT LCPDAT18={VEL 2.0,ACC 100.0,APO_DIST 100.0,APO_FAC 50.0,ORI_TYP #VAR,CIRC_TYP #BASE,JERK_FAC 50.0,EXAX_IGN 0}
DECL E6POS XP19={X 984.652771,Y 945.546021,Z 1250.39099,A -157.894501,B 46.0300903,C -166.346802,S 2,T 35,E1 0.0,E2 0.0,E3 0.0,E4 0.0,E5 0.0,E6 0.0}
DECL FDAT FP19={TOOL_NO 1,BASE_NO 0,IPO_FRAME #BASE,POINT2[] " ",TQ_STATE FALSE}
DECL LDAT LCPDAT19={VEL 2.0,ACC 100.0,APO_DIST 100.0,APO_FAC 50.0,ORI_TYP #VAR,CIRC_TYP #BASE,JERK_FAC 50.0,EXAX_IGN 0}
DECL E6POS XP20={X 984.663574,Y 955.53418,Z 1250.38696,A -157.897598,B 46.0290489,C -166.347504,S 2,T 35,E1 0.0,E2 0.0,E3 0.0,E4 0.0,E5 0.0,E6 0.0}
DECL FDAT FP20={TOOL_NO 1,BASE_NO 0,IPO_FRAME #BASE,POINT2[] " ",TQ_STATE FALSE}
DECL LDAT LCPDAT20={VEL 2.0,ACC 100.0,APO_DIST 100.0,APO_FAC 50.0,ORI_TYP #VAR,CIRC_TYP #BASE,JERK_FAC 50.0,EXAX_IGN 0}
DECL E6POS XP21={X 984.653503,Y 795.544006,Z 1251.38501,A -157.899902,B 46.0301018,C -166.3517,S 2,T 35,E1 0.0,E2 0.0,E3 0.0,E4 0.0,E5 0.0,E6 0.0}
DECL FDAT FP21={TOOL_NO 1,BASE_NO 0,IPO_FRAME #BASE,POINT2[] " ",TQ_STATE FALSE}
DECL LDAT LCPDAT21={VEL 2.0,ACC 100.0,APO_DIST 100.0,APO_FAC 50.0,ORI_TYP #VAR,CIRC_TYP #BASE,JERK_FAC 50.0,EXAX_IGN 0}
DECL E6POS XP22={X 984.650818,Y 845.544922,Z 1251.396,A -157.893295,B 46.0301704,C -166.345901,S 2,T 35,E1 0.0,E2 0.0,E3 0.0,E4 0.0,E5 0.0,E6 0.0}
DECL FDAT FP22={TOOL_NO 1,BASE_NO 0,IPO_FRAME #BASE,POINT2[] " ",TQ_STATE FALSE}
DECL LDAT LCPDAT22={VEL 2.0,ACC 100.0,APO_DIST 100.0,APO_FAC 50.0,ORI_TYP #VAR,CIRC_TYP #BASE,JERK_FAC 50.0,EXAX_IGN 0}
DECL E6POS XP23={X 984.651123,Y 945.543823,Z 1251.396,A -157.894302,B 46.0300789,C -166.346497,S 2,T 35,E1 0.0,E2 0.0,E3 0.0,E4 0.0,E5 0.0,E6 0.0}
DECL FDAT FP23={TOOL_NO 1,BASE_NO 0,IPO_FRAME #BASE,POINT2[] " ",TQ_STATE FALSE}
DECL LDAT LCPDAT23={VEL 2.0,ACC 100.0,APO_DIST 100.0,APO_FAC 50.0,ORI_TYP #VAR,CIRC_TYP #BASE,JERK_FAC 50.0,EXAX_IGN 0}
DECL E6POS XP24={X 984.664917,Y 955.530884,Z 1251.38794,A -157.8974,B 46.0288696,C -166.347107,S 2,T 35,E1 0.0,E2 0.0,E3 0.0,E4 0.0,E5 0.0,E6 0.0}
DECL FDAT FP24={TOOL_NO 1,BASE_NO 0,IPO_FRAME #BASE,POINT2[] " ",TQ_STATE FALSE}
DECL LDAT LCPDAT24={VEL 2.0,ACC 100.0,APO_DIST 100.0,APO_FAC 50.0,ORI_TYP #VAR,CIRC_TYP #BASE,JERK_FAC 50.0,EXAX_IGN 0}
DECL E6POS XP25={X 984.651306,Y 795.54248,Z 1252.38501,A -157.900894,B 46.0299797,C -166.3526,S 2,T 35,E1 0.0,E2 0.0,E3 0.0,E4 0.0,E5 0.0,E6 0.0}
DECL FDAT FP25={TOOL_NO 1,BASE_NO 0,IPO_FRAME #BASE,POINT2[] " ",TQ_STATE FALSE}
DECL LDAT LCPDAT25={VEL 2.0,ACC 100.0,APO_DIST 100.0,APO_FAC 50.0,ORI_TYP #VAR,CIRC_TYP #BASE,JERK_FAC 50.0,EXAX_IGN 0}
DECL E6POS XP26={X 984.650513,Y 845.543579,Z 1252.39697,A -157.893005,B 46.0300903,C -166.345398,S 2,T 35,E1 0.0,E2 0.0,E3 0.0,E4 0.0,E5 0.0,E6 0.0}
DECL FDAT FP26={TOOL_NO 1,BASE_NO 0,IPO_FRAME #BASE,POINT2[] " ",TQ_STATE FALSE}
DECL LDAT LCPDAT26={VEL 2.0,ACC 100.0,APO_DIST 100.0,APO_FAC 50.0,ORI_TYP #VAR,CIRC_TYP #BASE,JERK_FAC 50.0,EXAX_IGN 0}
DECL E6POS XP27={X 984.651489,Y 945.543579,Z 1252.39404,A -157.8936,B 46.0298805,C -166.345795,S 2,T 35,E1 0.0,E2 0.0,E3 0.0,E4 0.0,E5 0.0,E6 0.0}
DECL FDAT FP27={TOOL_NO 1,BASE_NO 0,IPO_FRAME #BASE,POINT2[] " ",TQ_STATE FALSE}
DECL LDAT LCPDAT27={VEL 2.0,ACC 100.0,APO_DIST 100.0,APO_FAC 50.0,ORI_TYP #VAR,CIRC_TYP #BASE,JERK_FAC 50.0,EXAX_IGN 0}
DECL E6POS XP28={X 984.665771,Y 955.527527,Z 1252.39099,A -157.8983,B 46.0289001,C -166.347595,S 2,T 35,E1 0.0,E2 0.0,E3 0.0,E4 0.0,E5 0.0,E6 0.0}
DECL FDAT FP28={TOOL_NO 1,BASE_NO 0,IPO_FRAME #BASE,POINT2[] " ",TQ_STATE FALSE}
DECL LDAT LCPDAT28={VEL 2.0,ACC 100.0,APO_DIST 100.0,APO_FAC 50.0,ORI_TYP #VAR,CIRC_TYP #BASE,JERK_FAC 50.0,EXAX_IGN 0}
DECL E6POS XP29={X 984.650085,Y 795.542297,Z 1253.38696,A -157.901505,B 46.0299797,C -166.353195,S 2,T 35,E1 0.0,E2 0.0,E3 0.0,E4 0.0,E5 0.0,E6 0.0}
DECL FDAT FP29={TOOL_NO 1,BASE_NO 0,IPO_FRAME #BASE,POINT2[] " ",TQ_STATE FALSE}
DECL LDAT LCPDAT29={VEL 2.0,ACC 100.0,APO_DIST 100.0,APO_FAC 50.0,ORI_TYP #VAR,CIRC_TYP #BASE,JERK_FAC 50.0,EXAX_IGN 0}
DECL E6POS XP30={X 984.648071,Y 845.544312,Z 1253.401,A -157.892197,B 46.0301208,C -166.344696,S 2,T 35,E1 0.0,E2 0.0,E3 0.0,E4 0.0,E5 0.0,E6 0.0}
DECL FDAT FP30={TOOL_NO 1,BASE_NO 0,IPO_FRAME #BASE,POINT2[] " ",TQ_STATE FALSE}
DECL LDAT LCPDAT30={VEL 2.0,ACC 100.0,APO_DIST 100.0,APO_FAC 50.0,ORI_TYP #VAR,CIRC_TYP #BASE,JERK_FAC 50.0,EXAX_IGN 0}
DECL E6POS XP31={X 984.648926,Y 945.543884,Z 1253.39905,A -157.893005,B 46.0299416,C -166.345306,S 2,T 35,E1 0.0,E2 0.0,E3 0.0,E4 0.0,E5 0.0,E6 0.0}
DECL FDAT FP31={TOOL_NO 1,BASE_NO 0,IPO_FRAME #BASE,POINT2[] " ",TQ_STATE FALSE}
DECL LDAT LCPDAT31={VEL 2.0,ACC 100.0,APO_DIST 100.0,APO_FAC 50.0,ORI_TYP #VAR,CIRC_TYP #BASE,JERK_FAC 50.0,EXAX_IGN 0}
DECL E6POS XP32={X 984.667603,Y 955.524109,Z 1253.39001,A -157.898804,B 46.0288582,C -166.347504,S 2,T 35,E1 0.0,E2 0.0,E3 0.0,E4 0.0,E5 0.0,E6 0.0}
DECL FDAT FP32={TOOL_NO 1,BASE_NO 0,IPO_FRAME #BASE,POINT2[] " ",TQ_STATE FALSE}
DECL LDAT LCPDAT32={VEL 2.0,ACC 100.0,APO_DIST 100.0,APO_FAC 50.0,ORI_TYP #VAR,CIRC_TYP #BASE,JERK_FAC 50.0,EXAX_IGN 0}
DECL E6POS XP33={X 984.648193,Y 795.539978,Z 1254.38599,A -157.902206,B 46.0296402,C -166.353394,S 2,T 35,E1 0.0,E2 0.0,E3 0.0,E4 0.0,E5 0.0,E6 0.0}
DECL FDAT FP33={TOOL_NO 1,BASE_NO 0,IPO_FRAME #BASE,POINT2[] " ",TQ_STATE FALSE}
DECL LDAT LCPDAT33={VEL 2.0,ACC 100.0,APO_DIST 100.0,APO_FAC 50.0,ORI_TYP #VAR,CIRC_TYP #BASE,JERK_FAC 50.0,EXAX_IGN 0}
DECL E6POS XP34={X 984.645325,Y 845.545105,Z 1254.40198,A -157.8918,B 46.0300484,C -166.344406,S 2,T 35,E1 0.0,E2 0.0,E3 0.0,E4 0.0,E5 0.0,E6 0.0}
DECL FDAT FP34={TOOL_NO 1,BASE_NO 0,IPO_FRAME #BASE,POINT2[] " ",TQ_STATE FALSE}
DECL LDAT LCPDAT34={VEL 2.0,ACC 100.0,APO_DIST 100.0,APO_FAC 50.0,ORI_TYP #VAR,CIRC_TYP #BASE,JERK_FAC 50.0,EXAX_IGN 0}
DECL E6POS XP35={X 984.64563,Y 945.544617,Z 1254.401,A -157.892395,B 46.0299911,C -166.345001,S 2,T 35,E1 0.0,E2 0.0,E3 0.0,E4 0.0,E5 0.0,E6 0.0}
DECL FDAT FP35={TOOL_NO 1,BASE_NO 0,IPO_FRAME #BASE,POINT2[] " ",TQ_STATE FALSE}
DECL LDAT LCPDAT35={VEL 2.0,ACC 100.0,APO_DIST 100.0,APO_FAC 50.0,ORI_TYP #VAR,CIRC_TYP #BASE,JERK_FAC 50.0,EXAX_IGN 0}
DECL E6POS XP36={X 984.668579,Y 955.521484,Z 1254.39099,A -157.8992,B 46.0287399,C -166.347794,S 2,T 35,E1 0.0,E2 0.0,E3 0.0,E4 0.0,E5 0.0,E6 0.0}
DECL FDAT FP36={TOOL_NO 1,BASE_NO 0,IPO_FRAME #BASE,POINT2[] " ",TQ_STATE FALSE}
DECL LDAT LCPDAT36={VEL 2.0,ACC 100.0,APO_DIST 100.0,APO_FAC 50.0,ORI_TYP #VAR,CIRC_TYP #BASE,JERK_FAC 50.0,EXAX_IGN 0}
DECL E6POS XP37={X 984.646729,Y 795.53833,Z 1255.38501,A -157.903,B 46.0293999,C -166.353806,S 2,T 35,E1 0.0,E2 0.0,E3 0.0,E4 0.0,E5 0.0,E6 0.0}
DECL FDAT FP37={TOOL_NO 1,BASE_NO 0,IPO_FRAME #BASE,POINT2[] " ",TQ_STATE FALSE}
DECL LDAT LCPDAT37={VEL 2.0,ACC 100.0,APO_DIST 100.0,APO_FAC 50.0,ORI_TYP #VAR,CIRC_TYP #BASE,JERK_FAC 50.0,EXAX_IGN 0}
DECL E6POS XP38={X 984.643677,Y 845.545593,Z 1255.40198,A -157.891098,B 46.0296898,C -166.343399,S 2,T 35,E1 0.0,E2 0.0,E3 0.0,E4 0.0,E5 0.0,E6 0.0}
DECL FDAT FP38={TOOL_NO 1,BASE_NO 0,IPO_FRAME #BASE,POINT2[] " ",TQ_STATE FALSE}
DECL LDAT LCPDAT38={VEL 2.0,ACC 100.0,APO_DIST 100.0,APO_FAC 50.0,ORI_TYP #VAR,CIRC_TYP #BASE,JERK_FAC 50.0,EXAX_IGN 0}
DECL E6POS XP39={X 984.643799,Y 945.544678,Z 1255.40198,A -157.891907,B 46.0297203,C -166.343994,S 2,T 35,E1 0.0,E2 0.0,E3 0.0,E4 0.0,E5 0.0,E6 0.0}
DECL FDAT FP39={TOOL_NO 1,BASE_NO 0,IPO_FRAME #BASE,POINT2[] " ",TQ_STATE FALSE}
DECL LDAT LCPDAT39={VEL 2.0,ACC 100.0,APO_DIST 100.0,APO_FAC 50.0,ORI_TYP #VAR,CIRC_TYP #BASE,JERK_FAC 50.0,EXAX_IGN 0}
DECL E6POS XP40={X 984.669128,Y 955.517517,Z 1255.39197,A -157.899307,B 46.0285683,C -166.347595,S 2,T 35,E1 0.0,E2 0.0,E3 0.0,E4 0.0,E5 0.0,E6 0.0}
DECL FDAT FP40={TOOL_NO 1,BASE_NO 0,IPO_FRAME #BASE,POINT2[] " ",TQ_STATE FALSE}
DECL LDAT LCPDAT40={VEL 2.0,ACC 100.0,APO_DIST 100.0,APO_FAC 50.0,ORI_TYP #VAR,CIRC_TYP #BASE,JERK_FAC 50.0,EXAX_IGN 0}
ENDDAT
